FUNCTION_BLOCK FB_FourthOrder
VAR_INPUT
END_VAR
VAR_OUTPUT
END_VAR
VAR CONSTANT
	order : INT := 4;
END_VAR

METHOD Cofactor : BOOL
VAR_INPUT
	ptrMatrix5x5	: POINTER TO ARRAY[1..5,1..5] OF LREAL;
	ptrCofactor		: POINTER TO LREAL;
	row				: INT;
	column			: INT;
END_VAR
VAR
	Matrix4x4	: ARRAY[1..4,1..4] OF LREAL;	
	i			: INT;
	j			: INT;
	k			: INT;
	m			: INT;
END_VAR
k := 1;
FOR i := 1 TO order+1 DO				// columns
	m := 1;
	IF i <> column THEN						
		FOR j := 1 TO order+1 DO		
			IF j <> row THEN
				Matrix4x4[k,m] := ptrMatrix5x5^[i,j];
				m := m + 1;
			END_IF
		END_FOR
		k := k + 1;
	END_IF
END_FOR

IF Determinant4x4(ptrDeterminant := ptrCofactor, ptrMatrix := ADR(Matrix4x4)) THEN
	Cofactor := TRUE;
ELSE
	Cofactor := FALSE;
END_IF
END_METHOD

METHOD Determinant4x4 : BOOL
VAR_INPUT
	ptrDeterminant	: POINTER TO LREAL;
	ptrMatrix		: POINTER TO ARRAY[1..4,1..4] OF LREAL;
END_VAR
VAR
	Matrix4x4		: ARRAY[1..4,1..4] OF LREAL;
	Element1		: LREAL;
	Element2		: LREAL;
	RowMultiplier	: LREAL;
	i				: INT;
	j				: INT;
	row 			: INT;
	currentRow		: INT;
	temp			: LREAL;
	Swap			: BOOL;
	index			: INT;
	found			: BOOL;
END_VAR
Matrix4x4 := ptrMatrix^;
Swap := FALSE;
FOR index := 1 TO 3 DO
	IF Matrix4x4[index,index] = 0 THEN
		found := FALSE;
		FOR i:=index+1 TO 4 DO
			IF Matrix4x4[index,i] <> 0 THEN
				row := i;
				found := TRUE;
				EXIT;
			END_IF
		END_FOR
		// swap current row with found row
		IF found THEN
			FOR i := 1 TO 4 DO
				temp := Matrix4x4[i,index];
				Matrix4x4[i,index] := Matrix4x4[i,row];
				Matrix4x4[i,row] := temp;
			END_FOR
			Swap := NOT Swap;
		ELSE
			ptrDeterminant^ := 0;
			Determinant4x4 := FALSE;
			RETURN;
		END_IF
	END_IF
	
	FOR j := index+1 TO 4 DO
		Element1 := Matrix4x4[index,index];
		Element2 := Matrix4x4[index,j];
		IF Element2 <> 0 THEN
			RowMultiplier := Element2/Element1;
			FOR i := 1 TO 4 DO
				Matrix4x4[i,j] := Matrix4x4[i,j] - RowMultiplier*Matrix4x4[i,index];
			END_FOR
		END_IF
	END_FOR
END_FOR

ptrDeterminant^ := 1;
FOR i := 1 TO 4 DO
	ptrDeterminant^ := ptrDeterminant^ * Matrix4x4[i,i];
END_FOR

IF Swap THEN
	ptrDeterminant^ := ptrDeterminant^ * (-1);
END_IF	
Determinant4x4 := TRUE;
END_METHOD

METHOD Determinant5x5 : BOOL
VAR_INPUT
	ptrDeterminant	: POINTER TO LREAL;
	ptrMatrix		: POINTER TO ARRAY[1..5,1..5] OF LREAL;
END_VAR
VAR
	Matrix5x5		: ARRAY[1..5,1..5] OF LREAL;
	Element1		: LREAL;
	Element2		: LREAL;
	RowMultiplier	: LREAL;
	i				: INT;
	j				: INT;
	row 			: INT;
	currentRow		: INT;
	temp			: LREAL;
	Swap			: BOOL;
	index			: INT;
	found			: BOOL;
END_VAR
Matrix5x5 := ptrMatrix^;
Swap := FALSE;
FOR index := 1 TO 4 DO
	IF Matrix5x5[index,index] = 0 THEN
		found := FALSE;
		FOR i:=index+1 TO 5 DO
			IF Matrix5x5[index,i] <> 0 THEN
				row := i;
				found := TRUE;
				EXIT;
			END_IF
		END_FOR
		// swap current row with found row
		IF found THEN
			FOR i := 1 TO 5 DO
				temp := Matrix5x5[i,index];
				Matrix5x5[i,index] := Matrix5x5[i,row];
				Matrix5x5[i,row] := temp;
			END_FOR
			Swap := NOT Swap;
		ELSE
			ptrDeterminant^ := 0;
			Determinant5x5 := FALSE;
			RETURN;
		END_IF
	END_IF
	
	FOR j := index+1 TO 5 DO
		Element1 := Matrix5x5[index,index];
		Element2 := Matrix5x5[index,j];
		IF Element2 <> 0 THEN
			RowMultiplier := Element2/Element1;
			FOR i := 1 TO 5 DO
				Matrix5x5[i,j] := Matrix5x5[i,j] - RowMultiplier*Matrix5x5[i,index];
			END_FOR
		END_IF
	END_FOR
END_FOR

ptrDeterminant^ := 1;
FOR i := 1 TO 5 DO
	ptrDeterminant^ := ptrDeterminant^ * Matrix5x5[i,i];
END_FOR

IF Swap THEN
	ptrDeterminant^ := ptrDeterminant^ * (-1);
END_IF	
Determinant5x5 := TRUE;
END_METHOD

METHOD FindCoefficients : BOOL
VAR_INPUT
	xValues		: POINTER TO ARRAY[1..GVL.NumberVisionPoints] OF LREAL;
	yValues		: POINTER TO ARRAY[1..GVL.NumberVisionPoints] OF LREAL;
	Coefficients: POINTER TO ARRAY[1..5] OF LREAL;
END_VAR
VAR_INST 
	xMatrix		: ARRAY[1..5, 1..GVL.NumberVisionPoints] OF LREAL;
	xTMatrix	: ARRAY[1..GVL.NumberVisionPoints, 1..5] OF LREAL; 
	xTxMatrix	: ARRAY[1..5,1..5] OF LREAL;
	xTxInverse	: ARRAY[1..5,1..5] OF LREAL;
	xTxXMatrix	: ARRAY[1..GVL.NumberVisionPoints,1..5] OF LREAL;
	xTyMatrix	: ARRAY[1..5] OF LREAL;
	i			: INT;
	j			: INT;
	k			: INT;
	DotProduct	: LREAL;
END_VAR
// fill out x matrix
// fill out transpose of x matrix
FOR i := 1 TO order+1 DO	// column
	FOR j := 1 TO GVL.NumberVisionPoints DO
		xMatrix[i,j] := EXPT((xValues^[j]),(i-1));	// column, row
		xTMatrix[j,i] := xMatrix[i,j];
	END_FOR
END_FOR

// fill out xT * x 
FOR i := 1 TO order+1 DO		// rows
	FOR j := 1 TO order+1 DO	
		DotProduct := 0;
		FOR k := 1 TO GVL.NumberVisionPoints DO
			DotProduct := DotProduct + xTMatrix[k,i]*xMatrix[j,k];
		END_FOR
		xTxMatrix[j,i] := DotProduct;
	END_FOR
END_FOR

// find out the inverse of xT*x
Inverse(ADR(xTxMatrix), ADR(xTxInverse));

// multiple xT*y
FOR i := 1 TO order+1 DO
	DotProduct := 0;
	FOR j := 1 TO GVL.NumberVisionPoints DO
		DotProduct := DotProduct + xTMatrix[j,i] * yValues^[j];
	END_FOR
	xTyMatrix[i] := DotProduct;
END_FOR

// multiply xTxInverse by xTy
FOR i := 1 TO order+1 DO
	DotProduct := 0;
	FOR j := 1 TO order+1 DO
		DotProduct := DotProduct + xTxInverse[j,i]*xTyMatrix[j];
	END_FOR
	Coefficients^[i] := DotProduct;
END_FOR
END_METHOD

METHOD FindYatX : BOOL
VAR_INPUT
	xValues			: POINTER TO ARRAY[1..GVL.NumberVisionPoints] OF LREAL;
	yValues			: POINTER TO ARRAY[1..GVL.NumberVisionPoints] OF LREAL;
	xPeak			: POINTER TO LREAL;
	yPeak			: POINTER TO LREAL;
END_VAR
VAR
	Coefficients	: ARRAY[1..5] OF LREAL;
END_VAR
FindCoefficients(xValues := xValues, yValues := yValues, Coefficients := ADR(Coefficients));
yPeak^ := Coefficients[1] + Coefficients[2] * xPeak^ + Coefficients[3]*EXPT(xPeak^,2) + 
		Coefficients[4]*EXPT(xPeak^,3) + Coefficients[5]*EXPT(xPeak^,4);
END_METHOD

METHOD Inverse : BOOL
VAR_INPUT
	ptrMatrix		: POINTER TO ARRAY[1..5,1..5] OF LREAL;
	ptrInverse		: POINTER TO ARRAY[1..5,1..5] OF LREAL;
END_VAR
VAR
	Determinant		: LREAL;
	Matrix			: ARRAY[1..5,1..5] OF LREAL;
	_Cofactor		: LREAL;
	i				: INT;
	j				: INT;
	SignRow: BOOL;
	SignColumn: BOOL;
END_VAR
IF Determinant5x5(ptrDeterminant := ADR(Determinant), ptrMatrix := ptrMatrix) THEN
	Determinant := 1 / Determinant;
	// get cofactors
	FOR i := 1 TO order+1 DO
		FOR j := 1 TO order+1 DO
			IF Cofactor(ptrMatrix5x5 := ptrMatrix, ptrCofactor := ADR(_Cofactor), row := i, column := j) THEN
				Matrix[i,j] := _Cofactor;
			ELSE
				Inverse := FALSE;
				RETURN;
			END_IF
		END_FOR
	END_FOR
	
	SignRow := TRUE;
	SignColumn := TRUE;
	FOR i := 1 TO order+1 DO
		FOR j := 1 TO order+1 DO
			IF NOT SignRow THEN
				Matrix[i,j] := (-1) * Matrix[i,j];
			END_IF
			SignRow := NOT SignRow;
		END_FOR
		SignColumn := NOT SignColumn;
		SignRow := SignColumn;
	END_FOR
	// transpose 
	Transpose(ADR(Matrix),ptrInverse);
	FOR i := 1 TO order+1 DO
		FOR j := 1 TO order+1 DO
			ptrInverse^[i,j] := Determinant * ptrInverse^[i,j];
		END_FOR
	END_FOR
	
	Inverse := TRUE;
ELSE
	Inverse := FALSE;
END_IF
END_METHOD

METHOD Transpose : BOOL
VAR_INPUT
	ptrMatrix		: POINTER TO ARRAY[1..5,1..5] OF LREAL;
	ptrTranspose	: POINTER TO ARRAY[1..5,1..5] OF LREAL;
END_VAR
VAR
	i				: INT;
	j				: INT;
END_VAR
FOR i := 1 TO order+1 DO
	FOR j := 1 TO order+1 DO
		ptrTranspose^[j,i] := ptrMatrix^[i,j];
	END_FOR
END_FOR
END_METHOD

END_FUNCTION_BLOCK

(* stored: Version 1.1.0.1, ProductVersion 3.1.4024.3
   POU FB_FourthOrder: Id {43f3b3e2-d85a-4949-b935-5ad920f6c56e}, SpecialFunc None
   Method Cofactor: Id {141795b6-f13f-4227-8263-340a87fcd5da}
   Method Determinant4x4: Id {e24d7971-7368-49a0-be38-a2dd669b6474}
   Method Determinant5x5: Id {e56af53c-ca7e-4072-84ad-5cb27504ee7a}
   Method FindCoefficients: Id {843de65b-dcbd-44fa-8e23-b40c74a2ae1d}
   Method FindYatX: Id {e166b935-2b01-4c4a-a248-6c9ccb60e316}
   Method Inverse: Id {431b774c-e7fd-4c28-b706-44889ff9860f}
   Method Transpose: Id {5863d92c-7668-40e1-9ce1-9449dbcdf8e5} *)
